FUNCTION_BLOCK Test_ReadWriteBySymbolName_KeepingHandle EXTENDS TUnitTestBase
VAR
    AdsReadWriteBySymbolName : TAdsReadWriteBySymbolName;
    TestInteger : TInteger;
    ReadWriteResult : INT;    
    ScanCount : DINT;
    State: INT;
END_VAR

CASE State OF
    0:
        TestInteger.Init(1111);
        ReadWriteResult := 0;
        ScanCount := 0;
    
        AdsReadWriteBySymbolName.Execute(
            AmsNetId:= '', 
            Port:= 851, 
            SymbolName:= 'PB_TestRunner.Test_ReadWriteBySymbolName_KeepingHandle.TestInteger#Inc', 
            ReadDataAddress:= ADR(ReadWriteResult), 
            ReadDataLength:= SIZEOF(ReadWriteResult), 
            WriteDataAddress:= 0, 
            WriteDataLength:= 0, 
            KeepSymbolHandle:= TRUE);

        Test_Started();
        State := 10;
        
    10:
        ScanCount := ScanCount + 1;
        IF NOT AdsReadWriteBySymbolName.Execution.Busy THEN
            State := 20;    
		END_IF
        
    20:
        Assertion.AssertEquals_INT(
            Expected     := 1112,
            Actual       := ReadWriteResult,
            ObjectName   := _TestName,
            Variablename := 'ReadWriteResult'); 
 
        Test_Finished();
        State := 0;
END_CASE

AdsReadWriteBySymbolName();

END_FUNCTION_BLOCK

(* stored: Version 1.1.0.1, ProductVersion 3.1.4024.3
   POU Test_ReadWriteBySymbolName_KeepingHandle: Id {ca782cb4-b471-010a-0158-4e11e9e53c17}, SpecialFunc None *)
